Staubli VAL3: getNumElements.pgx

public program getNumElements(num& x_nNumElems)
begin
  x_nNumElems = nElems
end
